// TIA Portal V20 export
DATA_BLOCK "DB_LaserOperation"   // DB431
// stored: AutoNumber false, InstanceOfName FB_LaserOperation, InstanceOfType FB
"FB_LaserOperation"
   // VAR
   //    sLaserTimeCh1 : "FB_TimeCounter";
   //    sLaserCycleTimeCh1 { S7_SetPoint := 'True'} : Int;
   // END_VAR
BEGIN
END_DATA_BLOCK
